// TIA Portal V20 export
ORGANIZATION_BLOCK "Startup"   // OB1015, LAD, Startup
TITLE = "Complete Restart"
// stored: AutoNumber false, Namespace Unit1.Em2, SetENOAutomatically false
   VAR_INPUT
      LostRetentive : Bool;   // True if retentive data are lost
      LostRTC : Bool;   // True if date and time are lost
   END_VAR
BEGIN

REGION Network 1 (SCL): Build the Absolut Reference Designator
   // Set the Absoult Reference Designator in the Config DB
   IF LEN(IN := "Unit1.Em2.Config".em.referenceDesignator.parent) <> 0 THEN
       "Unit1.Em2.Config".em.referenceDesignator.combined := CONCAT_WSTRING(IN1 := "Unit1.Em2.Config".em.referenceDesignator.parent, IN2 := WSTRING#'.', IN3 := "Unit1.Em2.Config".em.referenceDesignator.relative);
   ELSE
       "Unit1.Em2.Config".em.referenceDesignator.combined := "Unit1.Em2.Config".em.referenceDesignator.relative;
   END_IF;
END_REGION

REGION Network 2 (SCL): Assign axes data
   // Assign axes
   "Unit1.Em2.Config".axis[1] := "BA060AZSIDR1_JROutPnPLeftAxisX";
   "Unit1.Em2.Config".axis[2] := "BA060AZSIDR2_JROutPnPLeftAxisZ";
   "Unit1.Em2.Config".axis[3] := "BA060AZSIDR3_JROutPnPRightAxisX";
   "Unit1.Em2.Config".axis[4] := "BA060AZSIDR4_JROutPnPRightAxisZ";

   // FB Enable
   "Unit1.Em2.HmiInterface".cmJROutPnPLeftAxisX.commands.enableMasterControl := TRUE;
   "Unit1.Em2.HmiInterface".cmJROutPnPLeftAxisZ.commands.enableMasterControl := TRUE;
   "Unit1.Em2.HmiInterface".cmJROutPnPRightAxisX.commands.enableMasterControl := TRUE;
   "Unit1.Em2.HmiInterface".cmJROutPnPRightAxisZ.commands.enableMasterControl := TRUE;
END_REGION
END_ORGANIZATION_BLOCK
